// TwinCAT 3 PLC project ExerciseClickLog
// ProgramVersion: 3.1.4024.0
// libraries:
//   Tc2_Standard, * (Beckhoff Automation GmbH)
//   Tc2_System, * (Beckhoff Automation GmbH)
//   Tc3_Module, * (Beckhoff Automation GmbH)
// project tree:
//   / PlcTask.TcTTO
//   POUs/ FB_ClickLog.TcPOU, MAIN.TcPOU
// (motion and I/O tree: see PLC project checkerfunctions)
// real-time tasks:
//   TASK PlcTask: cycle T#10ms, priority 20, ADS port 350
//   TASK PlcTask1: cycle T#10ms, priority 21, ADS port 351
//   TASK PlcTask2: cycle T#10ms, priority 22, ADS port 352
//   TASK PlcTask3: cycle T#10ms, priority 23, ADS port 353
//   TASK PlcTask4: cycle T#10ms, priority 24, ADS port 354
//   TASK PlcTask5: cycle T#10ms, priority 25, ADS port 355
//   TASK PlcTask6: cycle T#10ms, priority 26, ADS port 356
//   TASK PlcTask7: cycle T#10ms, priority 27, ADS port 357

CONFIGURATION ExerciseClickLog
    RESOURCE PLC ON TwinCAT3
        TASK PlcTask(INTERVAL := T#10ms, PRIORITY := 22);
        PROGRAM MAIN WITH PlcTask : MAIN;
    END_RESOURCE
END_CONFIGURATION

// ---- POUs/MAIN.TcPOU
PROGRAM MAIN
VAR
myFB : FB_ClickLog;
minTime : TIME;
END_VAR

// NIET GETEST - CHATGPT GEMAAKT

myFB(); // Aanroepen van de FB in je programma
minTime := myFB.GetMinimumTime; // Haal de minimale tijd op

END_PROGRAM

// ---- POUs/FB_ClickLog.TcPOU
FUNCTION_BLOCK FB_ClickLog
VAR
    startTimer : BOOL := FALSE;
    clickDetected : BOOL;
    elapsedTime : TIME;
    timer : TON;
    clickTimes : ARRAY[1..50] OF TIME;
    clickIndex : INT := 0;
    pauseTimer : TON;
	InputVariable AT %I* : BOOL;
END_VAR

// NIET GETEST - CHATGPT GEMAAKT

IF NOT startTimer THEN
    IF InputVariable THEN // Vervang 'InputVariable' door je daadwerkelijke input
        startTimer := TRUE;
        timer.IN := TRUE;
        timer.PT := T#5s;
        pauseTimer.PT := T#2s;
    END_IF;
ELSE
    timer();
    pauseTimer();

    IF timer.Q THEN
        pauseTimer.IN := TRUE;
        timer.IN := FALSE;
    ELSIF pauseTimer.Q THEN
        pauseTimer.IN := FALSE;
        timer.IN := TRUE;
    END_IF;

    IF InputVariable AND NOT pauseTimer.Q THEN
        IF clickIndex < 10 THEN
            clickIndex := clickIndex + 1;
            clickTimes[clickIndex] := timer.ET;
        END_IF;
    END_IF;
END_IF;

// Reset timer elapsed time at the start of each recording period
IF timer.IN THEN
    timer.IN := FALSE;
    timer(); // Update de timer status
    timer.IN := TRUE;
END_IF;

METHOD GetMinimumTime : TIME
VAR_INPUT
	    i : INT;
END_VAR

// NIET GETEST - CHATGPT GEMAAKT
// controleer in welke formaat time word gezet in de clicktimes array
GetMinimumTime := T#24D; // Stel een hoge beginwaarde in

FOR i := 1 TO clickIndex DO
	IF clickTimes[i] < GetMinimumTime THEN
		GetMinimumTime := clickTimes[i];
	END_IF;
END_FOR;
END_METHOD

END_FUNCTION_BLOCK
